Fanuc KAREL source: CONT_TASK.kl

PROGRAM T
%NOLOCKGROUP
VAR
 v0 : STRING[40]
 v1 : INTEGER
BEGIN
 CONT_TASK(v0, v1)
END T
